FUNCTION_BLOCK Gradeamento (* Composite Function Block Type *)
  (* Standard: 61499-2 *)
  (* Version 0.0, 2/24/2026, template *)
  PACKAGE Hidryco.HidrycoLib;
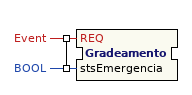
  EVENT_INPUT
    REQ WITH stsEmergencia;
  END_EVENT
  VAR_INPUT
    stsEmergencia : BOOL;
  END_VAR
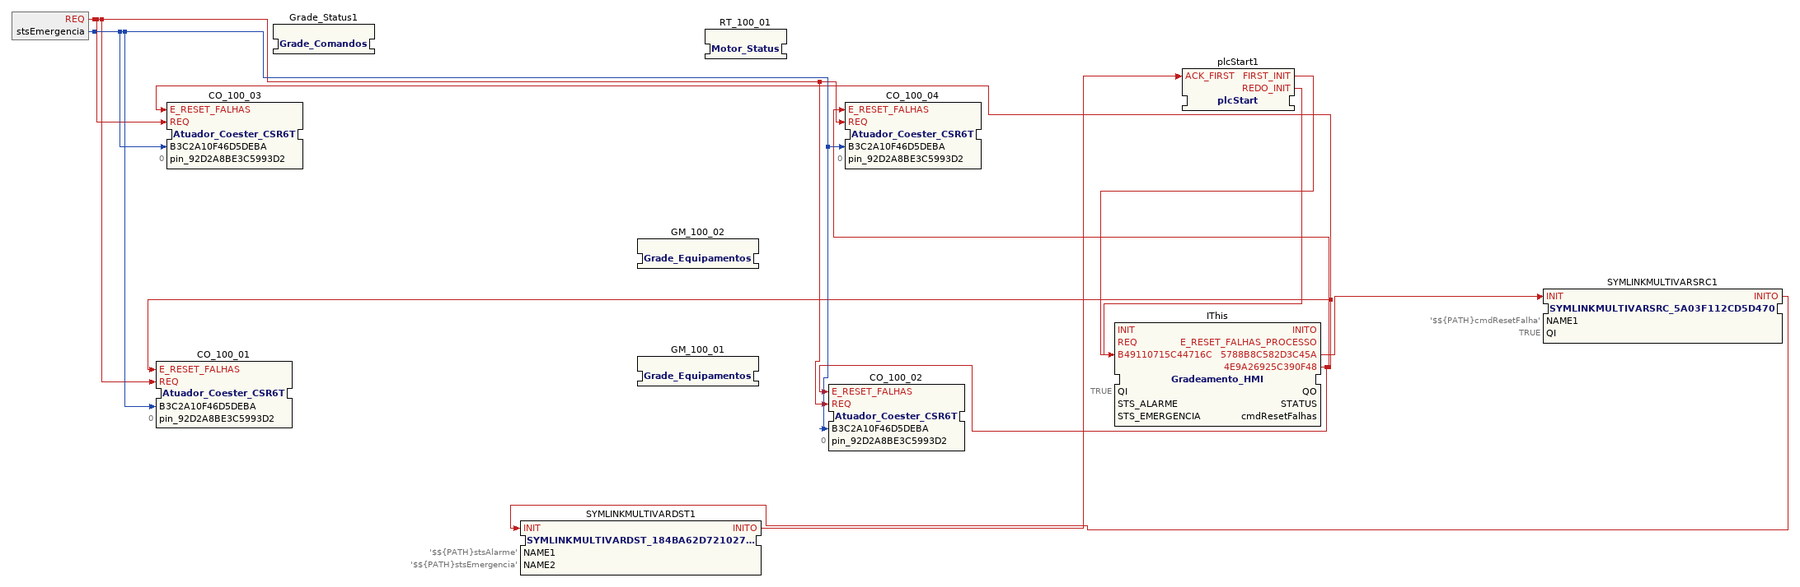
  FBS
    GM_100_02 : Grade_Equipamentos;
    GM_100_01 : Grade_Equipamentos;
    Grade_Status1 : Grade_Comandos;
    RT_100_01 : Motor_Status;
    SYMLINKMULTIVARSRC1 : SYMLINKMULTIVARSRC_5A03F112CD5D470(NAME1 := '$${PATH}cmdResetFalha', QI := TRUE); {SET_ATTRIBUTE(Configuration.GenericFBType.InterfaceParams, Runtime.System#I:=1;VALUE${I$}:INT)}
    plcStart1 : plcStart;
    IThis : Gradeamento_HMI(QI := TRUE);
    SYMLINKMULTIVARDST1 : SYMLINKMULTIVARDST_184BA62D721027C6E(NAME1 := '$${PATH}stsAlarme', NAME2 := '$${PATH}stsEmergencia'); {SET_ATTRIBUTE(Configuration.GenericFBType.InterfaceParams, Runtime.System#I:=2;VALUE${I$}:INT,INT)}
    CO_100_03 : Atuador_Coester_CSR6T(pin_92D2A8BE3C5993D2 := 0);
    CO_100_01 : Atuador_Coester_CSR6T(pin_92D2A8BE3C5993D2 := 0);
    CO_100_04 : Atuador_Coester_CSR6T(pin_92D2A8BE3C5993D2 := 0);
    CO_100_02 : Atuador_Coester_CSR6T(pin_92D2A8BE3C5993D2 := 0);
  END_FBS
  EVENT_CONNECTIONS
    SYMLINKMULTIVARDST1.INITO TO plcStart1.ACK_FIRST;
    SYMLINKMULTIVARSRC1.INITO TO SYMLINKMULTIVARDST1.INIT;
    plcStart1.FIRST_INIT TO IThis.B49110715C44716C;
    plcStart1.REDO_INIT TO IThis.B49110715C44716C;
    IThis.5788B8C582D3C45A TO SYMLINKMULTIVARSRC1.INIT;
    IThis.4E9A26925C390F48 TO CO_100_04.E_RESET_FALHAS;
    IThis.4E9A26925C390F48 TO CO_100_01.E_RESET_FALHAS;
    IThis.4E9A26925C390F48 TO CO_100_03.E_RESET_FALHAS;
    IThis.4E9A26925C390F48 TO CO_100_02.E_RESET_FALHAS;
    REQ TO CO_100_01.REQ;
    REQ TO CO_100_03.REQ;
    REQ TO CO_100_04.REQ;
    REQ TO CO_100_02.REQ;
  END_CONNECTIONS
  DATA_CONNECTIONS
    stsEmergencia TO CO_100_01.B3C2A10F46D5DEBA;
    stsEmergencia TO CO_100_03.B3C2A10F46D5DEBA;
    stsEmergencia TO CO_100_04.B3C2A10F46D5DEBA;
    stsEmergencia TO CO_100_02.B3C2A10F46D5DEBA;
  END_CONNECTIONS
END_FUNCTION_BLOCK
